(* IEC 61131-3 sources: AXOpen/src/simatic1500/ctrl/src, 7 files *)

(* ---- IDataEntity.st ---- *)
NAMESPACE ix.framework.data
    INTERFACE IDataEntity

    END_INTERFACE
END_NAMESPACE

(* ---- IDataExchange.st ---- *)
USING AXOpen.core;

NAMESPACE AXOpen.data
    INTERFACE IDataExchange
        METHOD Create : IIxTaskState
            VAR_INPUT
                Identifier : STRING[254];
            END_VAR
        END_METHOD

        METHOD Read : IIxTaskState
            VAR_INPUT
                Identifier : STRING[254];
            END_VAR
        END_METHOD

        METHOD Update : IIxTaskState
            VAR_INPUT
                Identifier : STRING[254];
            END_VAR
        END_METHOD

        METHOD Delete : IIxTaskState
            VAR_INPUT
                Identifier : STRING[254];
            END_VAR
        END_METHOD

        METHOD Restore
        END_METHOD
    END_INTERFACE
END_NAMESPACE

(* ---- DataEntity.st ---- *)
NAMESPACE AXOpen.data
    CLASS DataEntity IMPLEMENTS IDataEntity
        VAR PUBLIC
            {#ix-attr:[RenderIgnore("ShadowControl", "Control")]}
            DataEntityId : STRING[254];
        END_VAR
    END_CLASS
END_NAMESPACE

(* ---- DataExchange.st ---- *)
USING AXOpen.core;

NAMESPACE AXOpen.data
    CLASS DataExchange EXTENDS IxObject IMPLEMENTS IDataExchange
        VAR PUBLIC
           {#ix-set:AttributeName =  "<#Create#>"}
           CreateTask  : DataExchangeTask;
           {#ix-set:AttributeName =  "<#Read#>"}
           ReadTask    : DataExchangeTask;
           {#ix-set:AttributeName =  "<#Update#>"}
           UpdateTask  : DataExchangeTask;
           {#ix-set:AttributeName =  "<#Delete#>"}
           DeleteTask  : DataExchangeTask;
        END_VAR

        METHOD PRIVATE Run
            CreateTask.Initialize(THIS);
            ReadTask.Initialize(THIS);
            UpdateTask.Initialize(THIS);
            DeleteTask.Initialize(THIS);

            CreateTask.Execute();
            ReadTask.Execute();
            UpdateTask.Execute();
            DeleteTask.Execute();
        END_METHOD

        METHOD PUBLIC Run
            VAR_INPUT
                Parent : IIxObject;
            END_VAR
            THIS.Initialize(Parent);
            THIS.Run();
        END_METHOD

        METHOD PUBLIC Run
            VAR_INPUT
                Context : IIxContext;
            END_VAR
            THIS.Initialize(Context);
            THIS.Run();
        END_METHOD

        METHOD PUBLIC Create : IIxTaskState
            VAR_INPUT
                Identifier : STRING[254];
            END_VAR
            Create := CreateTask.Invoke(Identifier);
        END_METHOD

        METHOD PUBLIC Read : IIxTaskState
            VAR_INPUT
                Identifier : STRING[254];
            END_VAR
            Read := ReadTask.Invoke(Identifier);
        END_METHOD

        METHOD PUBLIC Update : IIxTaskState
            VAR_INPUT
                Identifier : STRING[254];
            END_VAR
            Update := UpdateTask.Invoke(Identifier);
        END_METHOD

        METHOD PUBLIC Delete : IIxTaskState
            VAR_INPUT
                Identifier : STRING[254];
            END_VAR
            Delete := DeleteTask.Invoke(Identifier);
        END_METHOD

        METHOD PUBLIC Restore
            CreateTask.Restore();
            ReadTask.Restore();
            UpdateTask.Restore();
            DeleteTask.Restore();
        END_METHOD
    END_CLASS
END_NAMESPACE

(* ---- DataExchangeTask.st ---- *)
USING AXOpen.core;
NAMESPACE AXOpen.data
    CLASS DataExchangeTask EXTENDS AXOpen.core.IxRemoteTask
        VAR PUBLIC
            DataEntityIdentifier : STRING[254];
        END_VAR

        METHOD PUBLIC Invoke : AXOpen.core.IIxTaskState
            VAR_INPUT
                identifier : STRING[254];
            END_VAR

            DataEntityIdentifier := identifier;
            Invoke := SUPER.Invoke();
        END_METHOD
    END_CLASS
END_NAMESPACE

(* ---- Rtc.st ---- *)
USING Siemens.Simatic.Clocks;
NAMESPACE AXOpen.S71500
    {S7.extern=ReadWrite}
    CLASS Rtc IMPLEMENTS AXOpen.Rtc.IAxoRtc
        METHOD PUBLIC NowUTC : LDATE_AND_TIME
            VAR_TEMP
                tmp_dt : LDATE_AND_TIME;
            END_VAR
            GetSystemDateTime(value => NowUTC);
        END_METHOD

        METHOD PUBLIC SetUTC : WORD
            VAR_INPUT
                Value : LDATE_AND_TIME;
            END_VAR
            SetUTC := SetSystemDateTime(value := Value);
        END_METHOD
    END_CLASS
END_NAMESPACE

(* ---- Rtm.st ---- *)
USING Siemens.Simatic.S71500.Clocks;
USING System.Timer;
NAMESPACE AXOpen.S71500
    {S7.extern=ReadWrite}
    CLASS Rtm IMPLEMENTS AXOpen.Rtm.IAxoRtm
        VAR
            _timer : OnDelay;
        END_VAR
        METHOD PUBLIC Elapsed : LTIME
            _timer(signal := TRUE, duration := LTIME#100000d2h4m8s16ms32ns);
            Elapsed := _timer.elapsedTime;
        END_METHOD
    END_CLASS
END_NAMESPACE
